// TIA Portal V19 export
FUNCTION_BLOCK "HMI_FB"   // FB50, LAD
TITLE = HMI Managment
AUTHOR : Piemme
FAMILY : System
// stored: Access Published, MemoryReserve 100, SetENOAutomatically false
   VAR
      FpReadClock : Bool;
   END_VAR
   VAR_TEMP
      ReturnValue : Int;
   END_VAR
   VAR CONSTANT
      "empty date" : DTL;
   END_VAR
   VAR_TEMP   // added for the SCL form of the ladder/FBD networks
      _w1 : Bool;
   END_VAR
BEGIN

REGION Network 1
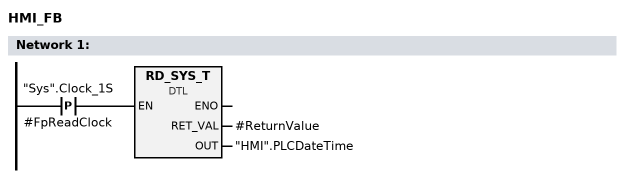
   RUNG wire#powerrail
      P_Contact(operand := "Sys".Clock_1S, bit := #FpReadClock)
      { S7_Templates := "date_type := DTL" } RD_SYS_T(RET_VAL => #ReturnValue, OUT => "HMI".PLCDateTime)
   END_RUNG
   // the same network as SCL:
   #_w1 := "Sys".Clock_1S AND NOT #FpReadClock;   // rising edge of "Sys".Clock_1S
   #FpReadClock := "Sys".Clock_1S;
   IF #_w1 THEN #ReturnValue := RD_SYS_T(OUT => "HMI".PLCDateTime); END_IF;
END_REGION

REGION Network 2 (SCL): Project Info
   (*
   "HMI".ProjectInfo.Job := '213123231';
   "HMI".ProjectInfo.Revision := 'V1.0';
   "HMI".ProjectInfo.RevisionDate := DTL#2022-09-13-00:00:00;
   "HMI".ProjectInfo.Programmer := 'DZN';
   "HMI".ProjectInfo.F_Signature := "RTG1SysInfo".F_SYSINFO.F_PROG_SIG;
   "HMI".ProjectInfo.F_CompilationDate := "RTG1SysInfo".F_SYSINFO.F_PROG_DAT;
   *)
END_REGION
END_FUNCTION_BLOCK
